FUNCTION_BLOCK CM_Actuator3State
VAR_INPUT
	CM_Number : INT;
	
	IN_MANUAL :BOOL;
	IN_HMI_HAND : BOOL;
	IN_AUTO : BOOL;
	
	IN_MANUAL_ON_1 : BOOL;
	IN_MANUAL_ON_2 : BOOL;
	
	IN_AUTO_ON_1 : BOOL;
	IN_AUTO_ON_2 : BOOL;
	
	IN_OFF : BOOL;
	
	IN_Alarm_Enable : BOOL;
	IN_CM_Alarm : BOOL;
	
	IN_CM_Interlock : BOOL;
END_VAR
VAR_OUTPUT
	AUTO_ON :BOOL;
	HMI_HAND_ON : BOOL;
	
	OUT_ON_1 : BOOL;
	OUT_ON_2 : BOOL;
	
	OUT_OFF :BOOL;
	
	PO_CM_Alarm : BOOL;
	
	PO_CM_Interlocked : BOOL;
END_VAR
VAR
	alarmDelay_H : systemTimeDelay;
	alarmDelay_L : systemTimeDelay;
END_VAR
VAR_IN_OUT
	CM_UDT_CTRL : Udt_CM_Actuator3State;
	Plant_control : Udt_PlantControl;
END_VAR

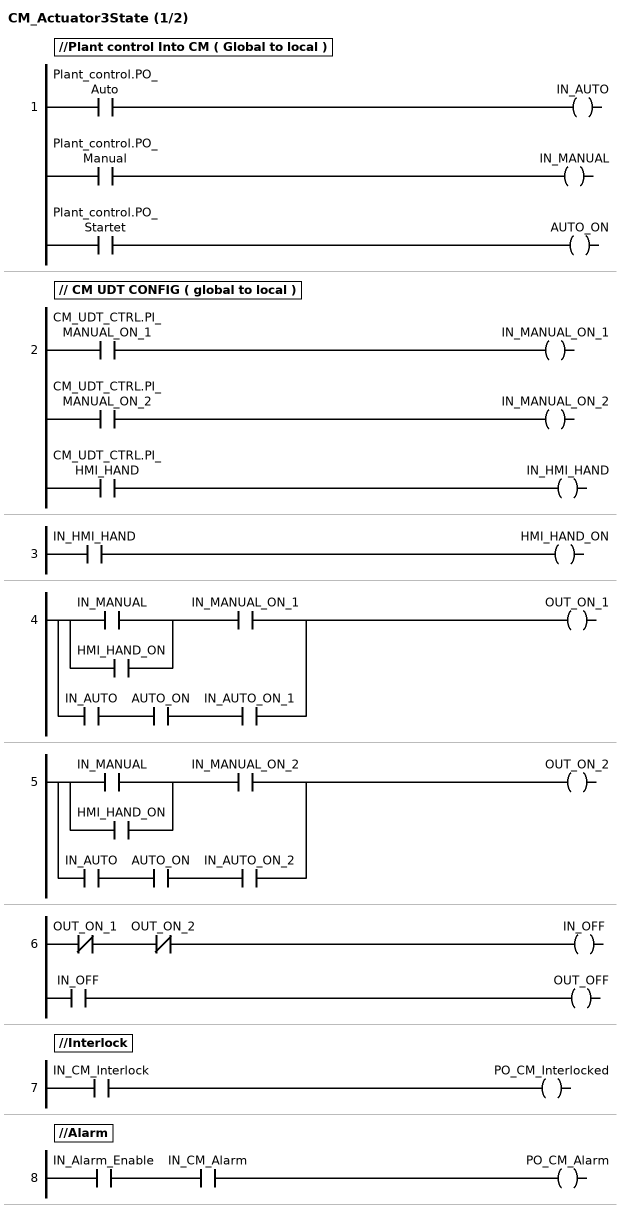
// NETWORK 1
// label: //Plant control Into CM ( Global to local )
IN_AUTO := Plant_control.PO_Auto;
IN_MANUAL := Plant_control.PO_Manual;
AUTO_ON := Plant_control.PO_Startet;

// NETWORK 2
// label: // CM UDT CONFIG ( global to local )
IN_MANUAL_ON_1 := CM_UDT_CTRL.PI_MANUAL_ON_1;
IN_MANUAL_ON_2 := CM_UDT_CTRL.PI_MANUAL_ON_2;
IN_HMI_HAND := CM_UDT_CTRL.PI_HMI_HAND;

// NETWORK 3
HMI_HAND_ON := IN_HMI_HAND;

// NETWORK 4
OUT_ON_1 := (IN_MANUAL OR HMI_HAND_ON) AND IN_MANUAL_ON_1 OR IN_AUTO AND AUTO_ON AND IN_AUTO_ON_1;

// NETWORK 5
OUT_ON_2 := (IN_MANUAL OR HMI_HAND_ON) AND IN_MANUAL_ON_2 OR IN_AUTO AND AUTO_ON AND IN_AUTO_ON_2;

// NETWORK 6
IN_OFF := NOT OUT_ON_1 AND NOT OUT_ON_2;
OUT_OFF := IN_OFF;

// NETWORK 7
// label: //Interlock
PO_CM_Interlocked := IN_CM_Interlock;

// NETWORK 8
// label: //Alarm
PO_CM_Alarm := IN_Alarm_Enable AND IN_CM_Alarm;

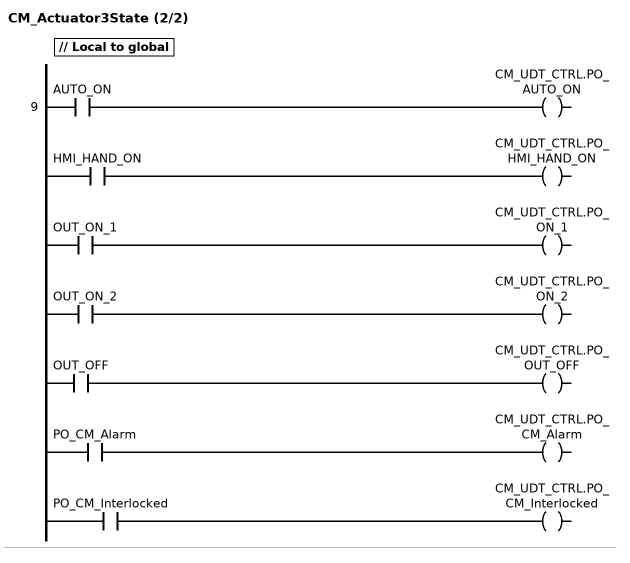
// NETWORK 9
// label: // Local to global
CM_UDT_CTRL.PO_AUTO_ON := AUTO_ON;
CM_UDT_CTRL.PO_HMI_HAND_ON := HMI_HAND_ON;
CM_UDT_CTRL.PO_ON_1 := OUT_ON_1;
CM_UDT_CTRL.PO_ON_2 := OUT_ON_2;
CM_UDT_CTRL.PO_OUT_OFF := OUT_OFF;
CM_UDT_CTRL.PO_CM_Alarm := PO_CM_Alarm;
CM_UDT_CTRL.PO_CM_Interlocked := PO_CM_Interlocked;

END_FUNCTION_BLOCK

(* stored: Version 1.1.0.1, ProductVersion 3.1.4024.13
   POU CM_Actuator3State: Id {2ab4e301-6d29-4071-b308-0e2f04923b4c}, SpecialFunc None *)
